PROGRAM general
VAR PERSISTENT
	//System date time function block
	system_date_time : date_time;
	//Daily reset bit, used throughout the program for any resets
	daily_reset : BOOL;
	//Alarm Acknoweldge unlatch timer
	alarm_ack_ton : ton;
	//Alarm Reset unlatch timer
	alarm_reset_ton : ton;
	//Alarm Ack and reset unlatch timer setpoint
	alarm_ack_unlatch_sp : TIME :=T#3s;
	
END_VAR

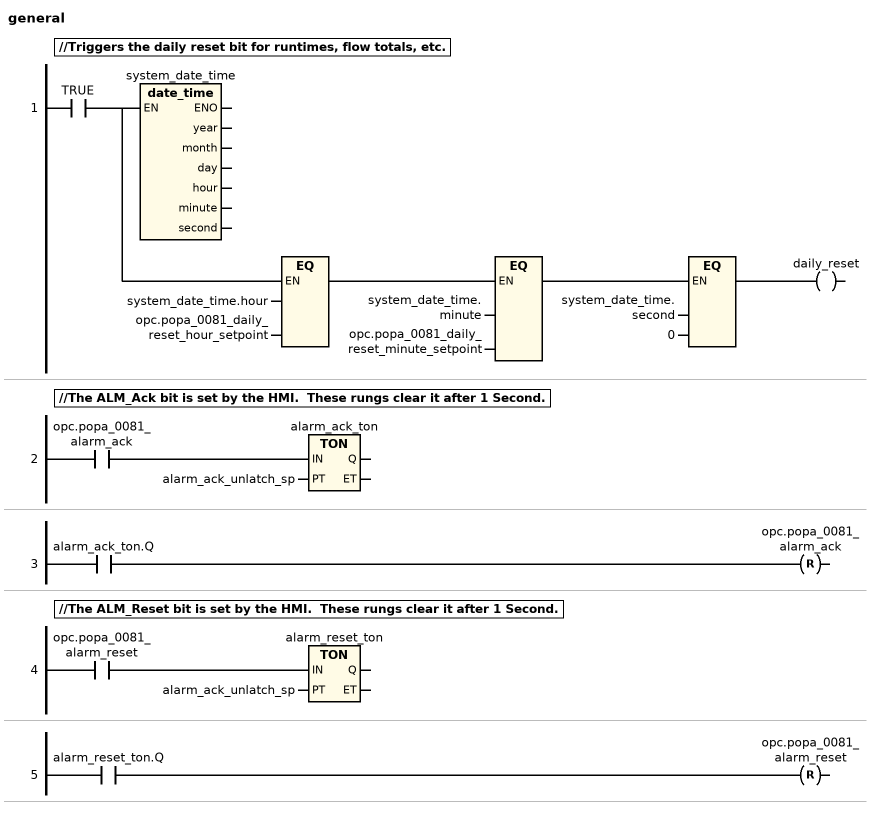
// NETWORK 1
// label: //Triggers the daily reset bit for runtimes, flow totals, etc.
system_date_time(); // date_time
daily_reset := system_date_time.hour = opc.popa_0081_daily_reset_hour_setpoint AND system_date_time.minute = opc.popa_0081_daily_reset_minute_setpoint AND system_date_time.second = 0;

// NETWORK 2
// label: //The ALM_Ack bit is set by the HMI.  These rungs clear it after 1 Second.
alarm_ack_ton(IN := opc.popa_0081_alarm_ack, PT := alarm_ack_unlatch_sp); // TON

// NETWORK 3
opc.popa_0081_alarm_ack R= alarm_ack_ton.Q;

// NETWORK 4
// label: //The ALM_Reset bit is set by the HMI.  These rungs clear it after 1 Second.
alarm_reset_ton(IN := opc.popa_0081_alarm_reset, PT := alarm_ack_unlatch_sp); // TON

// NETWORK 5
opc.popa_0081_alarm_reset R= alarm_reset_ton.Q;

END_PROGRAM

(* stored: Version 1.1.0.1, ProductVersion 3.1.4024.12
   POU general: Id {afd5554c-a122-45cd-a612-91df6056dfdf}, SpecialFunc None *)
